Omron CX-Programmer project 新工程 (CX-Programmer 9.73)

# PLC 新PLC1: CPM1(CPM1A) CPU30

## Program 新程序1 (no task)
; 项目概况 / 1．这个PLC程序实现了一个LED液压机的控制系统，控制液压机在LED灯具组装过程中的压制和成型工序。 / 2．系统通过启动按钮触发工作流程，支持手动和自动模式切换。 / 3．程序包含故障检测和保护功能，通过急停按钮停止设备运行，通过温度报警灯提示温度异常。 / 设备信息 / 1．系统包含启动按钮、急停按钮、手动/自动开关、模具闭合到位传感器、压力传感器和温度传感器。 / 2．执行器包括模具闭合阀、模具打开阀、液压机电机、压力控制阀和温度报警灯。 / 思路 / 1.操作员通过手动/自动开关选择运行模式，系统中自动模式标志和手动模式标志不可同时置位，以避免模式冲突。 / 2.系统通过手动/自动开关设置运行模式，手动模式用于操作员控制，自动模式用于系统自动流程。 / 3.在手动模式下，操作员通过按钮分别控制模具闭合阀、模具打开阀和液压机电机的启停。 / 4.在自动模式下，按下启动按钮后，系统首先激活模具闭合阀闭合模具，此时模具闭合阀和模具打开阀按顺序动作，以防止模具运动冲突。 / 5.模具闭合后，模具闭合到位传感器置位时，液压机电机才能启动，以确保安全压制。 / 6.压制过程中，压力传感器持续监测压力，若检测到异常，液压机电机停止，以避免设备损坏。 / 7.温度传感器监测温度，若温度异常，液压机电机停止。 / 8.温度异常时，温度报警灯亮起，以提示操作员。 / 9.压制完成后，系统激活模具打开阀打开模具。 / 10.为保障安全，若急停按钮按下，系统停止液压机电机、模具闭合阀和模具打开阀，以保护操作员和设备。

### Section 段1

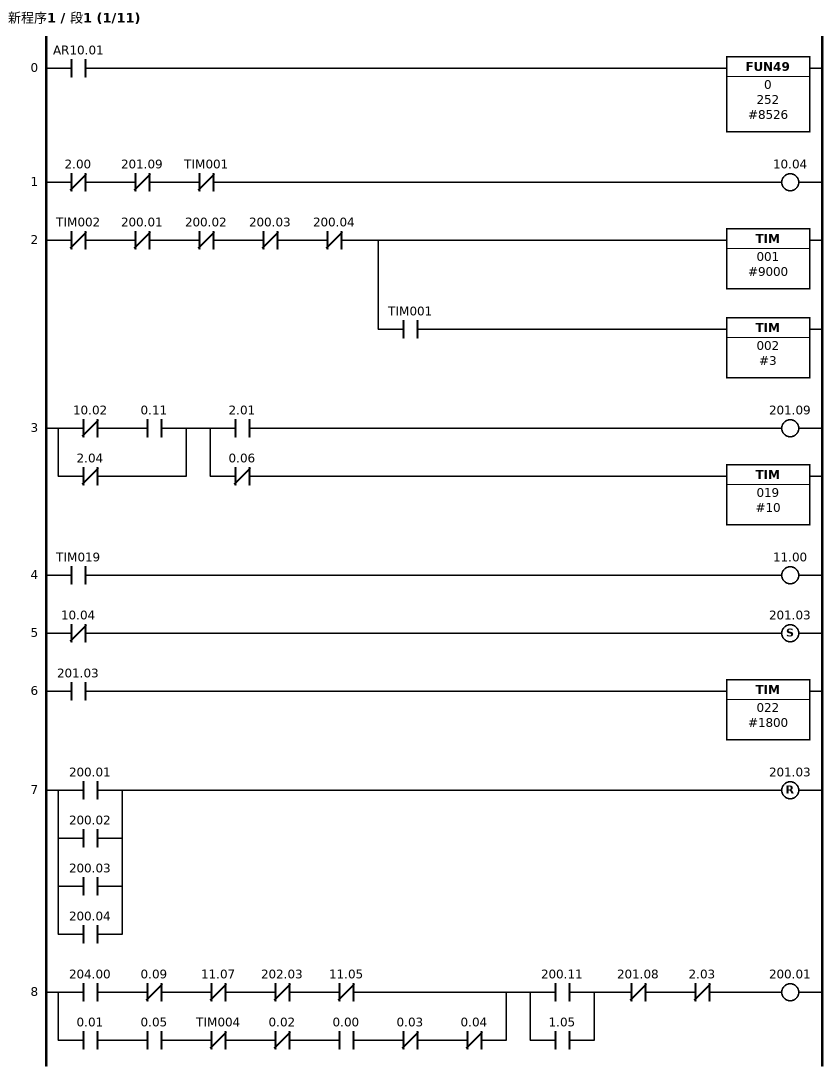
; rung 0
LD AR10.01
FUN49 0 252 #8526
; rung 1
LDNOT 2.00
ANDNOT 201.09
ANDNOT TIM001
OUT 10.04
; rung 2
LDNOT TIM002
ANDNOT 200.01
ANDNOT 200.02
ANDNOT 200.03
ANDNOT 200.04
TIM 001 #9000
AND TIM001
TIM 002 #3
; rung 3
LDNOT 10.02
AND 0.11
ORNOT 2.04
OUT TR0
AND 2.01
OUT 201.09
LD TR0
ANDNOT 0.06
TIM 019 #10
; rung 4
LD TIM019
OUT 11.00
; rung 5
LDNOT 10.04
SET 201.03
; rung 6
LD 201.03
TIM 022 #1800
; rung 7
LD 200.01
OR 200.02
OR 200.03
OR 200.04
RSET 201.03
; rung 8
LD 204.00
ANDNOT 0.09
ANDNOT 11.07
ANDNOT 202.03
ANDNOT 11.05
LD 0.01
AND 0.05
ANDNOT TIM004
ANDNOT 0.02
AND 0.00
ANDNOT 0.03
ANDNOT 0.04
ORLD
LD 200.11
OR 1.05
ANDLD
ANDNOT 201.08
ANDNOT 2.03
OUT 200.01

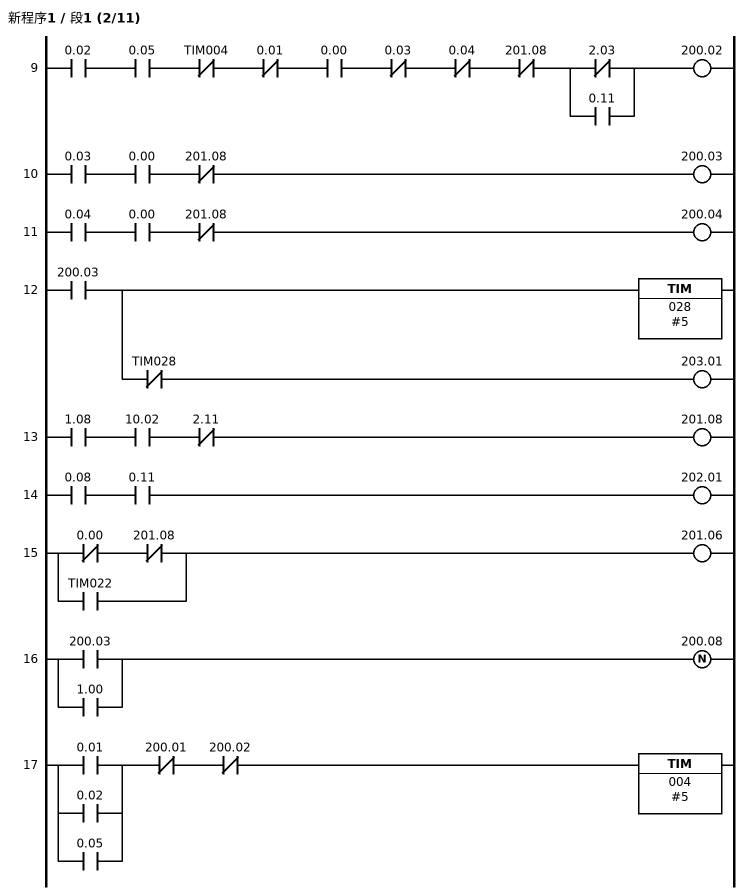
; rung 9
LD 0.02
AND 0.05
ANDNOT TIM004
ANDNOT 0.01
AND 0.00
ANDNOT 0.03
ANDNOT 0.04
ANDNOT 201.08
LDNOT 2.03
OR 0.11
ANDLD
OUT 200.02
; rung 10
LD 0.03
AND 0.00
ANDNOT 201.08
OUT 200.03
; rung 11
LD 0.04
AND 0.00
ANDNOT 201.08
OUT 200.04
; rung 12
LD 200.03
TIM 028 #5
ANDNOT TIM028
OUT 203.01
; rung 13
LD 1.08
AND 10.02
ANDNOT 2.11
OUT 201.08
; rung 14
LD 0.08
AND 0.11
OUT 202.01
; rung 15
LDNOT 0.00
ANDNOT 201.08
OR TIM022
OUT 201.06
; rung 16
LD 200.03
OR 1.00
DIFD(14) 200.08
; rung 17
LD 0.01
OR 0.02
OR 0.05
ANDNOT 200.01
ANDNOT 200.02
TIM 004 #5

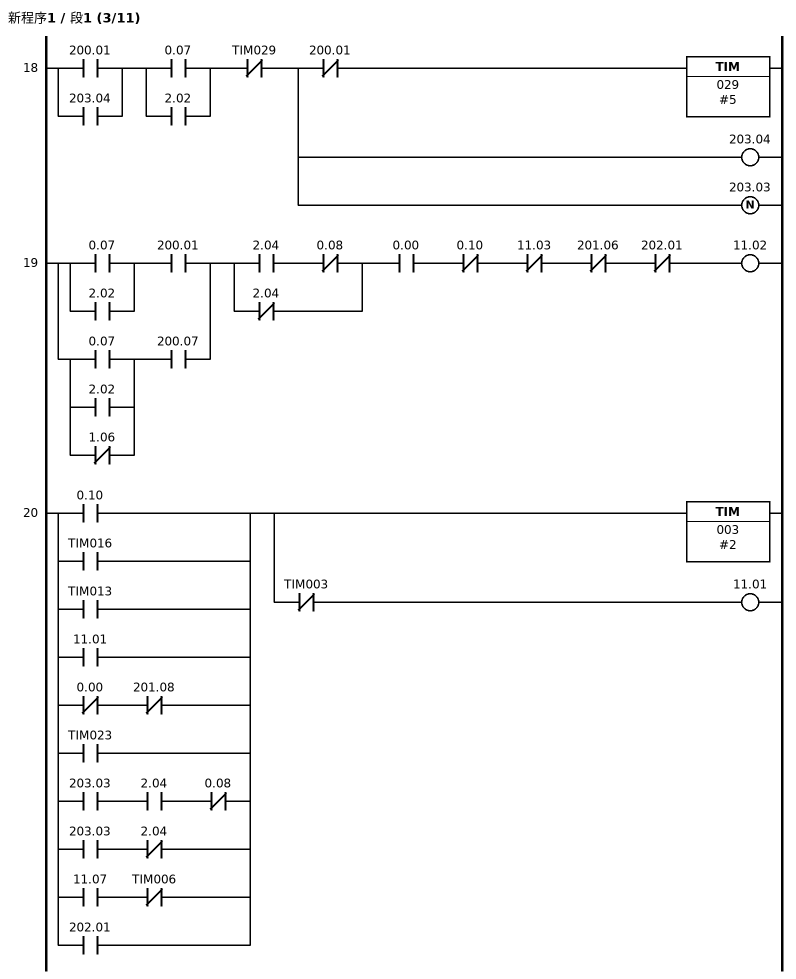
; rung 18
LD 200.01
OR 203.04
LD 0.07
OR 2.02
ANDLD
ANDNOT TIM029
OUT TR0
ANDNOT 200.01
TIM 029 #5
LD TR0
OUT 203.04
DIFD(14) 203.03
; rung 19
LD 0.07
OR 2.02
AND 200.01
LD 0.07
OR 2.02
ORNOT 1.06
AND 200.07
ORLD
LD 2.04
ANDNOT 0.08
ORNOT 2.04
ANDLD
AND 0.00
ANDNOT 0.10
ANDNOT 11.03
ANDNOT 201.06
ANDNOT 202.01
OUT 11.02
; rung 20
LD 0.10
OR TIM016
OR TIM013
OR 11.01
LDNOT 0.00
ANDNOT 201.08
ORLD
OR TIM023
LD 203.03
AND 2.04
ANDNOT 0.08
ORLD
LD 203.03
ANDNOT 2.04
ORLD
LD 11.07
ANDNOT TIM006
ORLD
OR 202.01
TIM 003 #2
ANDNOT TIM003
OUT 11.01

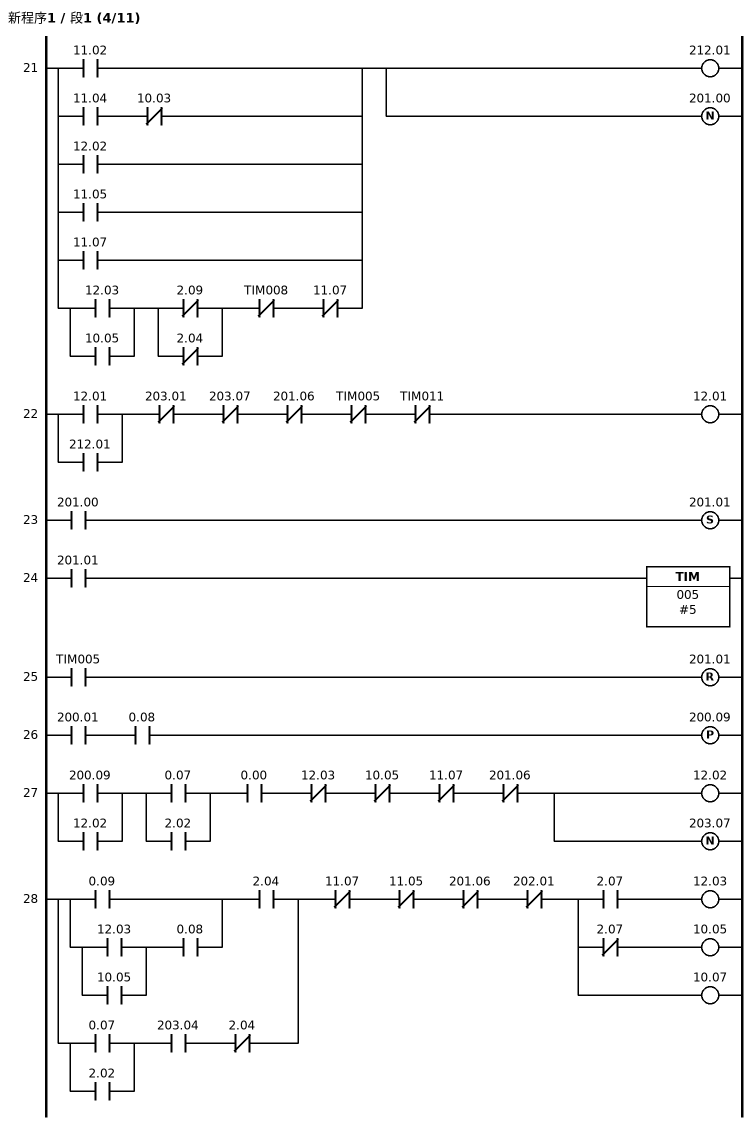
; rung 21
LD 11.02
LD 11.04
ANDNOT 10.03
ORLD
OR 12.02
OR 11.05
OR 11.07
LD 12.03
OR 10.05
LDNOT 2.09
ORNOT 2.04
ANDLD
ANDNOT TIM008
ANDNOT 11.07
ORLD
OUT 212.01
DIFD(14) 201.00
; rung 22
LD 12.01
OR 212.01
ANDNOT 203.01
ANDNOT 203.07
ANDNOT 201.06
ANDNOT TIM005
ANDNOT TIM011
OUT 12.01
; rung 23
LD 201.00
SET 201.01
; rung 24
LD 201.01
TIM 005 #5
; rung 25
LD TIM005
RSET 201.01
; rung 26
LD 200.01
AND 0.08
DIFU(13) 200.09
; rung 27
LD 200.09
OR 12.02
LD 0.07
OR 2.02
ANDLD
AND 0.00
ANDNOT 12.03
ANDNOT 10.05
ANDNOT 11.07
ANDNOT 201.06
OUT 12.02
DIFD(14) 203.07
; rung 28
LD 0.09
LD 12.03
OR 10.05
AND 0.08
ORLD
AND 2.04
LD 0.07
OR 2.02
AND 203.04
ANDNOT 2.04
ORLD
ANDNOT 11.07
ANDNOT 11.05
ANDNOT 201.06
ANDNOT 202.01
OUT TR0
AND 2.07
OUT 12.03
LD TR0
ANDNOT 2.07
OUT 10.05
LD TR0
OUT 10.07

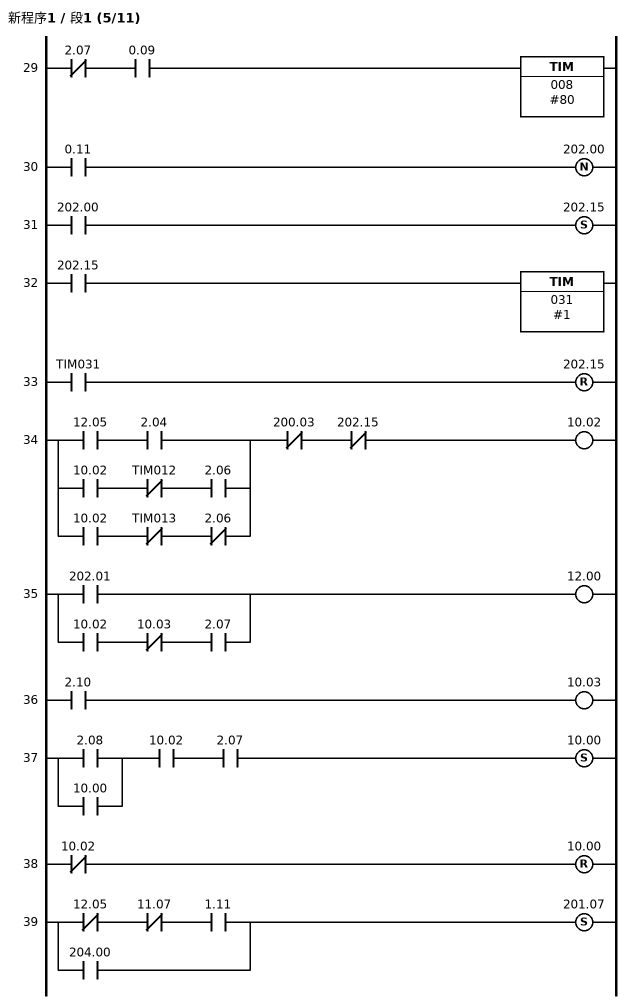
; rung 29
LDNOT 2.07
AND 0.09
TIM 008 #80
; rung 30
LD 0.11
DIFD(14) 202.00
; rung 31
LD 202.00
SET 202.15
; rung 32
LD 202.15
TIM 031 #1
; rung 33
LD TIM031
RSET 202.15
; rung 34
LD 12.05
AND 2.04
LD 10.02
ANDNOT TIM012
AND 2.06
ORLD
LD 10.02
ANDNOT TIM013
ANDNOT 2.06
ORLD
ANDNOT 200.03
ANDNOT 202.15
OUT 10.02
; rung 35
LD 202.01
LD 10.02
ANDNOT 10.03
AND 2.07
ORLD
OUT 12.00
; rung 36
LD 2.10
OUT 10.03
; rung 37
LD 2.08
OR 10.00
AND 10.02
AND 2.07
SET 10.00
; rung 38
LDNOT 10.02
RSET 10.00
; rung 39
LDNOT 12.05
ANDNOT 11.07
AND 1.11
OR 204.00
SET 201.07

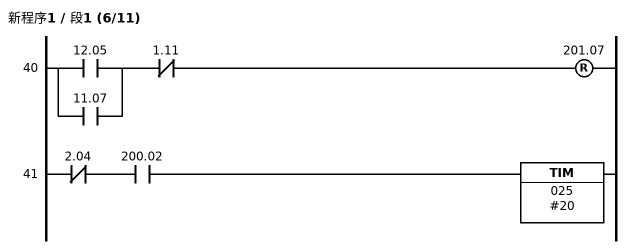
; rung 40
LD 12.05
OR 11.07
ANDNOT 1.11
RSET 201.07
; rung 41
LDNOT 2.04
AND 200.02
TIM 025 #20

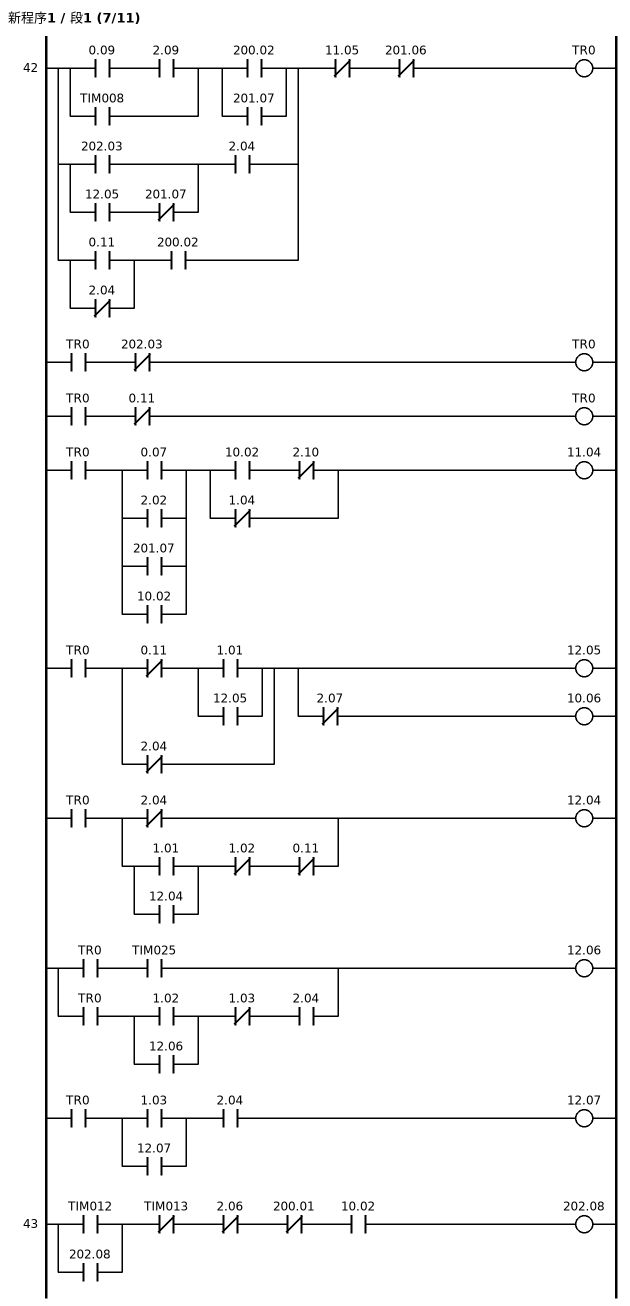
; rung 42
LD 0.09
AND 2.09
OR TIM008
LD 200.02
OR 201.07
ANDLD
LD 202.03
LD 12.05
ANDNOT 201.07
ORLD
AND 2.04
ORLD
LD 0.11
ORNOT 2.04
AND 200.02
ORLD
ANDNOT 11.05
ANDNOT 201.06
OUT TR0
LD 0.07
OR 2.02
OR 201.07
OR 10.02
ANDLD
LD 10.02
ANDNOT 2.10
ORNOT 1.04
ANDLD
OUT 11.04
LD TR0
ANDNOT 202.03
OUT TR0
LDNOT 0.11
LD 1.01
OR 12.05
ANDLD
ORNOT 2.04
ANDLD
OUT 12.05
ANDNOT 2.07
OUT 10.06
LD TR0
LDNOT 2.04
LD 1.01
OR 12.04
ANDNOT 1.02
ANDNOT 0.11
ORLD
ANDLD
OUT 12.04
LD TR0
AND TIM025
LD TR0
ANDNOT 0.11
OUT TR0
LD 1.02
OR 12.06
ANDLD
ANDNOT 1.03
AND 2.04
ORLD
OUT 12.06
LD TR0
LD 1.03
OR 12.07
ANDLD
AND 2.04
OUT 12.07
; rung 43
LD TIM012
OR 202.08
ANDNOT TIM013
ANDNOT 2.06
ANDNOT 200.01
AND 10.02
OUT 202.08

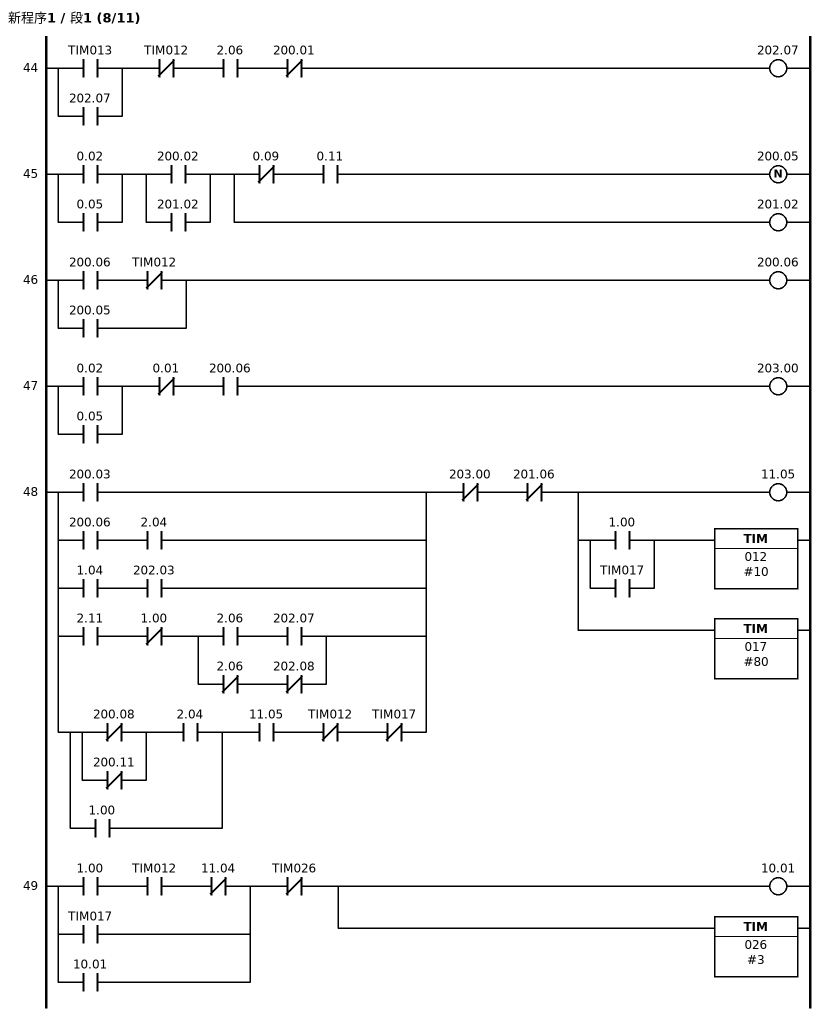
; rung 44
LD TIM013
OR 202.07
ANDNOT TIM012
AND 2.06
ANDNOT 200.01
OUT 202.07
; rung 45
LD 0.02
OR 0.05
LD 200.02
OR 201.02
ANDLD
OUT TR0
ANDNOT 0.09
AND 0.11
DIFD(14) 200.05
LD TR0
OUT 201.02
; rung 46
LD 200.06
ANDNOT TIM012
OR 200.05
OUT 200.06
; rung 47
LD 0.02
OR 0.05
ANDNOT 0.01
AND 200.06
OUT 203.00
; rung 48
LD 200.03
LD 200.06
AND 2.04
ORLD
LD 1.04
AND 202.03
ORLD
LD 2.11
ANDNOT 1.00
LD 2.06
AND 202.07
LDNOT 2.06
ANDNOT 202.08
ORLD
ANDLD
ORLD
LDNOT 200.08
ORNOT 200.11
AND 2.04
OR 1.00
AND 11.05
ANDNOT TIM012
ANDNOT TIM017
ORLD
ANDNOT 203.00
ANDNOT 201.06
OUT TR0
OUT 11.05
LD 1.00
OR TIM017
ANDLD
TIM 012 #10
LD TR0
TIM 017 #80
; rung 49
LD 1.00
AND TIM012
ANDNOT 11.04
OR TIM017
OR 10.01
ANDNOT TIM026
OUT 10.01
TIM 026 #3

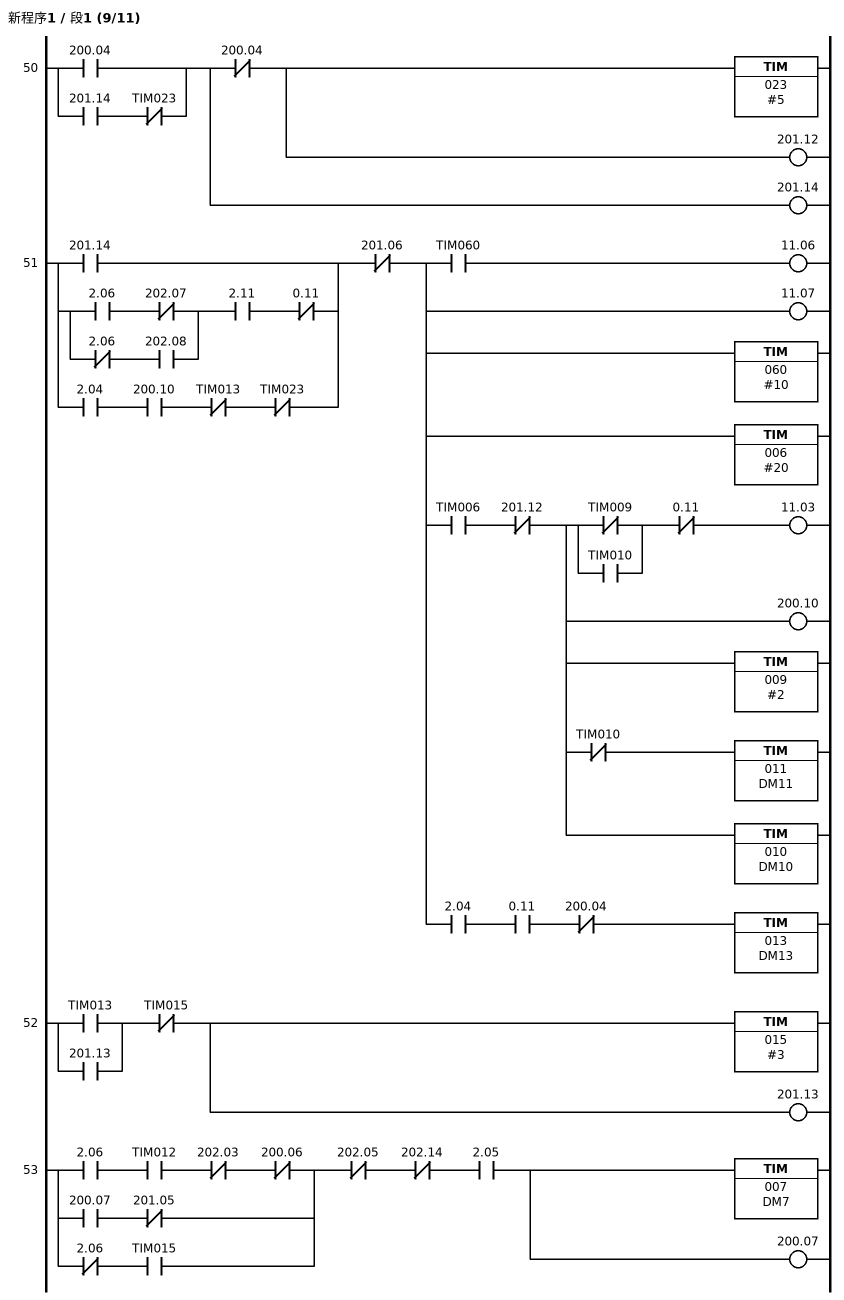
; rung 50
LD 200.04
LD 201.14
ANDNOT TIM023
ORLD
OUT TR0
ANDNOT 200.04
TIM 023 #5
OUT 201.12
LD TR0
OUT 201.14
; rung 51
LD 201.14
LD 2.06
ANDNOT 202.07
LDNOT 2.06
AND 202.08
ORLD
AND 2.11
ANDNOT 0.11
ORLD
LD 2.04
AND 200.10
ANDNOT TIM013
ANDNOT TIM023
ORLD
ANDNOT 201.06
OUT TR0
AND TIM060
OUT 11.06
LD TR0
OUT 11.07
TIM 060 #10
TIM 006 #20
AND TIM006
ANDNOT 201.12
OUT TR1
LDNOT TIM009
OR TIM010
ANDLD
ANDNOT 0.11
OUT 11.03
LD TR1
OUT 200.10
TIM 009 #2
ANDNOT TIM010
TIM 011 DM11
LD TR1
TIM 010 DM10
LD TR0
AND 2.04
AND 0.11
ANDNOT 200.04
TIM 013 DM13
; rung 52
LD TIM013
OR 201.13
ANDNOT TIM015
TIM 015 #3
OUT 201.13
; rung 53
LD 2.06
AND TIM012
ANDNOT 202.03
ANDNOT 200.06
LD 200.07
ANDNOT 201.05
ORLD
LDNOT 2.06
AND TIM015
ORLD
ANDNOT 202.05
ANDNOT 202.14
AND 2.05
TIM 007 DM7
OUT 200.07

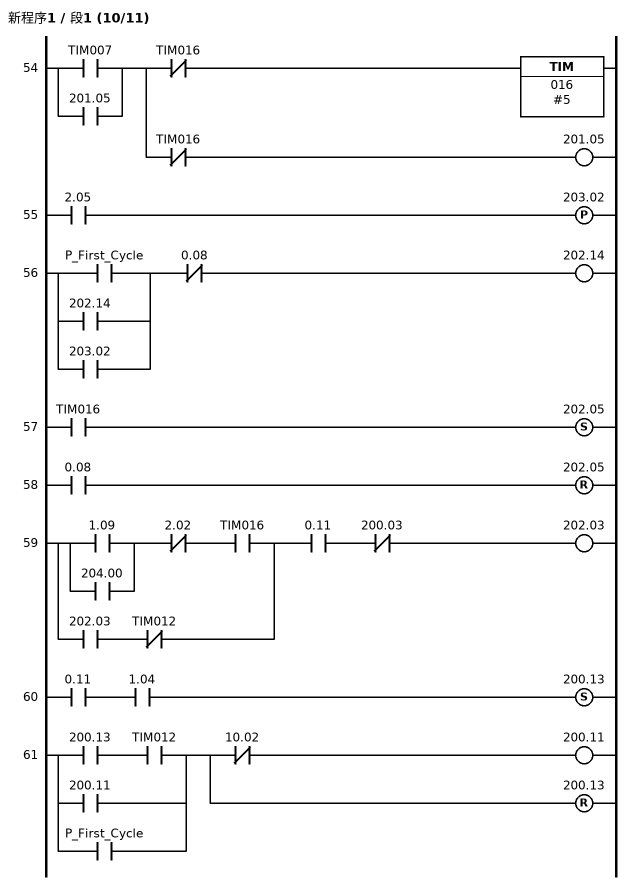
; rung 54
LD TIM007
OR 201.05
OUT TR0
ANDNOT TIM016
TIM 016 #5
LD TR0
ANDNOT TIM016
OUT 201.05
; rung 55
LD 2.05
DIFU(13) 203.02
; rung 56
LD P_First_Cycle
OR 202.14
OR 203.02
ANDNOT 0.08
OUT 202.14
; rung 57
LD TIM016
SET 202.05
; rung 58
LD 0.08
RSET 202.05
; rung 59
LD 1.09
OR 204.00
ANDNOT 2.02
AND TIM016
LD 202.03
ANDNOT TIM012
ORLD
AND 0.11
ANDNOT 200.03
OUT 202.03
; rung 60
LD 0.11
AND 1.04
SET 200.13
; rung 61
LD 200.13
AND TIM012
OR 200.11
OR P_First_Cycle
OUT TR0
ANDNOT 10.02
OUT 200.11
LD TR0
RSET 200.13

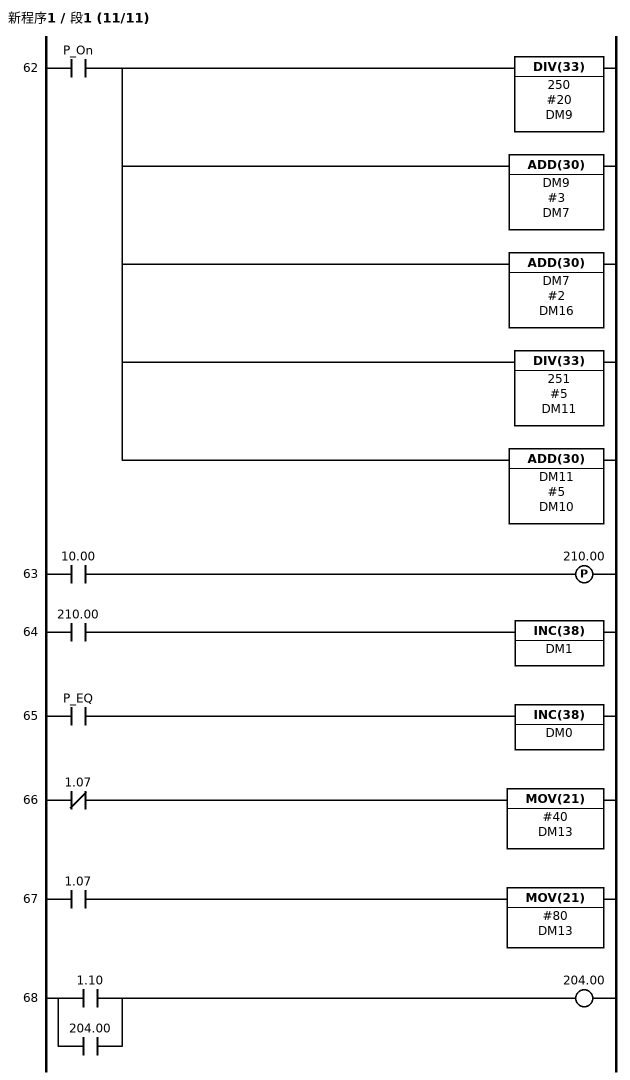
; rung 62
LD P_On
DIV(33) 250 #20 DM9
ADD(30) DM9 #3 DM7
ADD(30) DM7 #2 DM16
DIV(33) 251 #5 DM11
ADD(30) DM11 #5 DM10
; rung 63
LD 10.00
DIFU(13) 210.00
; rung 64
LD 210.00
INC(38) DM1
; rung 65
LD P_EQ
INC(38) DM0
; rung 66
LDNOT 1.07
MOV(21) #40 DM13
; rung 67
LD 1.07
MOV(21) #80 DM13
; rung 68
LD 1.10
OR 204.00
OUT 204.00
; rung 69
END(01)